Staubli VAL3: get.pgx

public program get(string& x_sItem[], num x_nIndex)
  local num l_nSize
  local string l_sKey
  local num i
begin
  x_sItem=sKey[x_nIndex]
end
